// TIA Portal V21 export
FUNCTION "Main zone" : Void   // FC35, LAD
{ S7_Optimized_Access := 'TRUE' }
// stored: SetENOAutomatically false
   VAR_TEMP
      NonUsato : Bool;
   END_VAR
   VAR CONSTANT
      Nessuna : Int := 0;
   END_VAR
BEGIN
END_FUNCTION
